Staubli VAL3: combineString.pgx

public program combineString(string x_sInput)
  local num l_nElement
begin

  for l_nElement = 0 to size(x_sInput)-1
  endFor

end
